// TIA Portal V17 export
// export: Created 2023-02-13T11:16:04.3967979Z, ExportSetting WithDefaults, DisplayName Totally Integrated Automation Portal, DisplayVersion V17, DisplayName TIA Portal Openness, DisplayVersion V17, DisplayName TIA Portal Teamcenter Gateway, DisplayVersion V17, DisplayName TIA Portal Version Control Interface, DisplayVersion V17, DisplayName SINAMICS Startdrive Advanced, DisplayVersion V17, DisplayName SINAMICS Startdrive G130, G150, S120, S150, SINAMICS MV, S210, DisplayVersion V17, DisplayName SINAMICS Startdrive G110M, G120, G120C, G120D, G120P, G115D, DisplayVersion V17, DisplayName STEP 7 Professional, DisplayVersion V17, DisplayName STEP 7 Safety, DisplayVersion V17, DisplayName WinCC Professional, DisplayVersion V17
DATA_BLOCK "Osa to MB"   // DB264
{ S7_Optimized_Access := 'FALSE' }
VERSION : 0.1
// stored: AutoNumber false, DBAccessibleFromOPCUA true, DBAccessibleFromWebserver true, IsOnlyStoredInLoadMemory false, IsWriteProtectedInAS false
   VAR
      HeartBeat : Bool;   // Clock 1hz
      Product_Ready : Bool;
      Product_LineOpen : Bool;
      Product_SupplyON : Bool;
      Product_Transfer_Complete : Bool;
      freeBool5 : Bool;
      freeBool6 : Bool;
      freeBool7 : Bool;
      freeBool8 : Bool;
      freeBool9 : Bool;
      freeBool10 : Bool;
      freeBool11 : Bool;
      freeBool12 : Bool;
      freeBool13 : Bool;
      freeBool14 : Bool;
      freeBool15 : Bool;
      freeBool16 : Bool;
      freeBool17 : Bool;
      freeBool18 : Bool;
      freeBool19 : Bool;
      freeBool20 : Bool;
      freeBool21 : Bool;
      freeBool22 : Bool;
      freeBool23 : Bool;
   END_VAR
BEGIN
END_DATA_BLOCK
